// TIA Portal V18 export
ORGANIZATION_BLOCK "Startup"   // OB100, LAD, Startup
TITLE = "Complete Restart"
{ S7_Optimized_Access := 'TRUE' }
VERSION : 0.1
// stored: AutoNumber true, IsIECCheckEnabled false, SetENOAutomatically false
   VAR_INPUT
      LostRetentive : Bool;   // True if retentive data are lost
      LostRTC : Bool;   // True if date and time are lost
   END_VAR
BEGIN

REGION Network 1
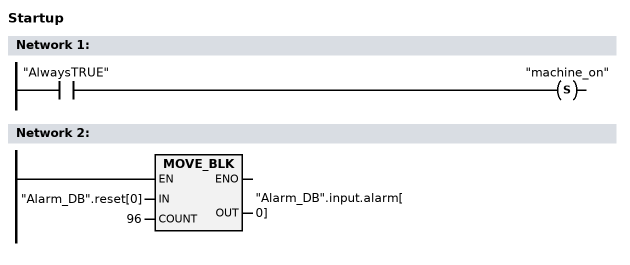
   RUNG wire#powerrail
      Contact( "AlwaysTRUE" )
      S_Coil( "machine_on" )
   END_RUNG
   // the same network as SCL:
   IF "AlwaysTRUE" THEN "machine_on" := TRUE; END_IF;
END_REGION

REGION Network 2
   MOVE_BLK(IN := "Alarm_DB".reset[0], COUNT := 96, OUT => "Alarm_DB".input.alarm[0]);
END_REGION
END_ORGANIZATION_BLOCK
